TYPE ST_MODBUS_SEND_FRAME :
STRUCT
	StartAddress:WORD;
	sendQuantity:WORD;
	SendData:ARRAY [0..10] OF WORD;
END_STRUCT
END_TYPE

(* stored: Version 1.1.0.1
   DUT ST_MODBUS_SEND_FRAME: Id {82330ffd-2e7f-4137-b7d8-97f0aa437904} *)
